FUNCTION_BLOCK Variable_Control_Mapping_Model
VAR_INPUT
	Controller_Leg_Variable	: ARRAY[1..18] OF LREAL;		// 控制模型中的驱动器位置
END_VAR
VAR_OUTPUT
	Model_Leg_Variable	: ARRAY[1..18] OF LREAL;		// 六足机构模型中的腿位置
END_VAR
VAR
END_VAR

Model_Leg_Variable[1]		:= Controller_Leg_Variable[2];
Model_Leg_Variable[2]		:= Controller_Leg_Variable[3];
Model_Leg_Variable[3]		:= Controller_Leg_Variable[1];
Model_Leg_Variable[4]		:= Controller_Leg_Variable[17];
Model_Leg_Variable[5]		:= Controller_Leg_Variable[18];
Model_Leg_Variable[6]		:= Controller_Leg_Variable[16];
Model_Leg_Variable[7]		:= Controller_Leg_Variable[14];
Model_Leg_Variable[8]		:= Controller_Leg_Variable[15];
Model_Leg_Variable[9]		:= Controller_Leg_Variable[13];
Model_Leg_Variable[10]		:= Controller_Leg_Variable[11];
Model_Leg_Variable[11]		:= Controller_Leg_Variable[12];
Model_Leg_Variable[12]		:= Controller_Leg_Variable[10];
Model_Leg_Variable[13]		:= Controller_Leg_Variable[8];
Model_Leg_Variable[14]		:= Controller_Leg_Variable[9];
Model_Leg_Variable[15]		:= Controller_Leg_Variable[7];
Model_Leg_Variable[16]		:= Controller_Leg_Variable[5];
Model_Leg_Variable[17]		:= Controller_Leg_Variable[6];
Model_Leg_Variable[18]		:= Controller_Leg_Variable[4];

END_FUNCTION_BLOCK

(* stored: Version 1.1.0.1, ProductVersion 3.1.4020.12
   POU Variable_Control_Mapping_Model: Id {9d48883c-8b80-4f05-b48f-637a56faf3fc}, SpecialFunc None *)
